# EPICS autosave request: stdApp/Db/recordPV_settings.req
$(P)$(Q)$(R).INP
$(P)$(Q)$(R).SCAN
$(P)$(Q)$(R)
